FUNCTION F_Error : DWORD
VAR_INPUT
	Error_Code															: DWORD;
	Error_On															: BOOL;
	Error																: INT;
END_VAR
VAR
	Error_Bit															: DWORD;
END_VAR

// F_Error - If Error is true, Error_Code is 
// Rev 1.0 - September 24, 2024

Error_Bit																:= LREAL_TO_DWORD(EXPT(2, Error));
F_Error																	:= SEL(Error_On, Error_Code AND NOT Error_Bit, Error_Code OR Error_Bit);

END_FUNCTION

(* stored: Version 1.1.0.1, ProductVersion 3.1.4024.13
   POU F_Error: Id {adab9405-bb83-4095-bfe1-ac83aa121e65}, SpecialFunc None *)
